{attribute addProperty BoxType "EP2339-0021-0017"}
{attribute addProperty Id "ChannelAT %I*ARRAY[0..15] OF Channel_E4AEF59E128160Channel_1AT %Q*ARRAY[0..15] OF Channel_7F374EB0128160WcStateAT %I*WcState_F855686C1620InfoDataAT %I*InfoData_2EA224846480"}
{attribute addProperty CRC "1354158181"}
{attribute addProperty SizeInBites "336"}
{attribute addProperty SizeInBytes "42"}
TYPE EP2339_067D5D8B :
STRUCT
	{attribute addProperty Name "Channel"}
	Channel : ARRAY[0..15] OF Channel_E4AEF59E;
	{attribute addProperty Name "Channel_1"}
	Channel_1 : ARRAY[0..15] OF Channel_7F374EB0;
	{attribute addProperty Name "WcState"}
	WcState : WcState_F855686C;
	{attribute addProperty Name "InfoData"}
	InfoData : InfoData_2EA22484;
END_STRUCT
END_TYPE

(* stored: Version 1.2.0.0, ProductVersion 3.1.4024.9
   DUT EP2339_067D5D8B: Id {346d2525-9796-4048-b32c-c4b0dac360bc} *)
